Yaskawa INFORM job: test1_robodk.jbi

/JOB
//NAME Hexagon
//POS
///NPOS 620,0,0,0,0,0
///TOOL 9
///POSTYPE PULSE
///PULSE
C00000=-4,42,-30,0,-18,-176
C00001=-4,48,-28,0,-14,-176
C00002=-1,49,-25,0,-16,-179
C00003=-1,52,-18,0,-19,-179
C00004=-4,54,-14,0,-22,-176
C00005=-7,53,-17,0,-20,-173
C00006=-7,50,-24,0,-16,-173
C00007=-4,48,-28,0,-14,-176
C00008=-4,48,-28,0,-14,-176
C00009=-4,48,-28,0,-14,-176
C00010=-4,48,-28,0,-14,-176
C00011=-1,49,-25,0,-16,-179
C00012=-1,52,-18,0,-19,-179
C00013=-4,54,-15,0,-21,-176
C00014=-7,53,-18,0,-20,-173
C00015=-7,50,-24,0,-16,-173
C00016=-4,48,-28,0,-14,-176
C00017=-4,48,-28,0,-14,-176
C00018=-1,49,-25,0,-16,-179
C00019=-1,49,-25,0,-16,-179
C00020=-1,49,-25,0,-15,-179
C00021=-1,49,-25,0,-16,-179
C00022=-2,49,-26,0,-15,-178
C00023=-2,49,-26,0,-15,-178
C00024=-2,49,-26,0,-15,-178
C00025=-1,50,-25,0,-16,-179
C00026=-1,50,-24,0,-16,-179
C00027=-2,49,-26,0,-15,-178
C00028=-2,49,-26,0,-15,-178
C00029=-2,49,-26,0,-15,-178
C00030=-1,50,-24,0,-16,-179
C00031=-1,50,-24,0,-16,-179
C00032=-3,49,-27,0,-15,-177
C00033=-3,49,-27,0,-15,-177
C00034=-3,49,-27,0,-15,-177
C00035=-1,50,-24,0,-16,-179
C00036=-1,50,-24,0,-16,-179
C00037=-3,48,-27,0,-14,-177
C00038=-3,48,-27,0,-14,-177
C00039=-4,48,-27,0,-14,-176
C00040=-1,50,-23,0,-17,-179
C00041=-1,50,-23,0,-17,-179
C00042=-4,48,-28,0,-14,-176
C00043=-4,48,-28,0,-14,-176
C00044=-4,48,-28,0,-14,-176
C00045=-1,50,-23,0,-17,-179
C00046=-1,50,-23,0,-17,-179
C00047=-4,48,-28,0,-14,-176
C00048=-4,48,-28,0,-14,-176
C00049=-1,50,-22,0,-17,-179
C00050=-1,51,-22,0,-17,-179
C00051=-5,48,-28,0,-14,-175
C00052=-5,48,-28,0,-14,-175
C00053=-1,51,-22,0,-17,-179
C00054=-1,51,-22,0,-17,-179
C00055=-5,48,-28,0,-14,-175
C00056=-5,48,-28,0,-14,-175
C00057=-1,51,-22,0,-18,-179
C00058=-1,51,-21,0,-18,-179
C00059=-5,48,-28,0,-14,-175
C00060=-5,48,-27,0,-14,-175
C00061=-1,51,-21,0,-18,-179
C00062=-1,51,-21,0,-18,-179
C00063=-5,48,-27,0,-14,-175
C00064=-5,48,-27,0,-14,-175
C00065=-1,51,-21,0,-18,-179
C00066=-1,51,-21,0,-18,-179
C00067=-5,48,-27,0,-14,-175
C00068=-5,48,-27,0,-14,-175
C00069=-1,51,-20,0,-18,-179
C00070=-1,51,-20,0,-18,-179
C00071=-5,49,-27,0,-14,-175
C00072=-5,49,-27,0,-15,-175
C00073=-1,52,-20,0,-19,-179
C00074=-1,52,-20,0,-19,-179
C00075=-5,49,-27,0,-15,-175
C00076=-5,49,-27,0,-15,-175
C00077=-1,52,-19,0,-19,-179
C00078=-1,52,-19,0,-19,-179
C00079=-5,49,-27,0,-15,-175
C00080=-6,49,-27,0,-15,-174
C00081=-1,52,-19,0,-19,-179
C00082=-1,52,-19,0,-19,-179
C00083=-6,49,-26,0,-15,-174
C00084=-6,49,-26,0,-15,-174
C00085=-1,52,-19,0,-19,-179
C00086=-1,52,-18,0,-19,-179
C00087=-6,49,-26,0,-15,-174
C00088=-6,49,-26,0,-15,-174
C00089=-1,52,-18,0,-19,-179
C00090=-1,52,-18,0,-19,-179
C00091=-6,49,-26,0,-15,-174
C00092=-6,49,-26,0,-15,-174
C00093=-1,52,-18,0,-20,-179
C00094=-1,52,-18,0,-20,-179
C00095=-6,49,-26,0,-15,-174
C00096=-6,49,-26,0,-15,-174
C00097=-2,52,-18,0,-20,-178
C00098=-2,52,-18,0,-20,-178
C00099=-6,49,-26,0,-15,-174
C00100=-6,49,-26,0,-15,-174
C00101=-2,52,-18,0,-20,-178
C00102=-2,52,-18,0,-20,-178
C00103=-6,49,-26,0,-15,-174
C00104=-6,49,-26,0,-15,-174
C00105=-2,53,-18,0,-20,-178
C00106=-2,53,-18,0,-20,-178
C00107=-6,49,-25,0,-15,-174
C00108=-6,49,-25,0,-15,-174
C00109=-2,53,-18,0,-20,-178
C00110=-2,53,-17,0,-20,-178
C00111=-7,49,-25,0,-16,-173
C00112=-7,49,-25,0,-16,-173
C00113=-2,53,-17,0,-20,-178
C00114=-2,53,-17,0,-20,-178
C00115=-7,49,-25,0,-16,-173
C00116=-7,49,-25,0,-16,-173
C00117=-2,53,-17,0,-20,-178
C00118=-2,53,-17,0,-20,-178
C00119=-7,49,-25,0,-16,-173
C00120=-7,49,-25,0,-16,-173
C00121=-2,53,-17,0,-20,-178
C00122=-2,53,-17,0,-20,-178
C00123=-7,49,-25,0,-16,-173
C00124=-7,50,-25,0,-16,-173
C00125=-2,53,-17,0,-20,-178
C00126=-3,53,-17,0,-20,-177
C00127=-7,50,-24,0,-16,-173
C00128=-7,50,-24,0,-16,-173
C00129=-3,53,-17,0,-20,-177
C00130=-3,53,-17,0,-20,-177
C00131=-7,50,-24,0,-16,-173
C00132=-7,50,-24,0,-16,-173
C00133=-3,53,-16,0,-20,-177
C00134=-3,53,-16,0,-21,-177
C00135=-7,50,-24,0,-16,-173
C00136=-7,50,-24,0,-16,-173
C00137=-3,53,-16,0,-21,-177
C00138=-3,53,-16,0,-21,-177
C00139=-7,50,-24,0,-16,-173
C00140=-7,50,-23,0,-17,-173
C00141=-3,53,-16,0,-21,-177
C00142=-3,53,-16,0,-21,-177
C00143=-7,50,-23,0,-17,-173
C00144=-7,50,-23,0,-17,-173
C00145=-3,53,-16,0,-21,-177
C00146=-3,53,-16,0,-21,-177
C00147=-7,50,-23,0,-17,-173
C00148=-7,50,-22,0,-17,-173
C00149=-3,53,-16,0,-21,-177
C00150=-3,53,-16,0,-21,-177
C00151=-7,51,-22,0,-17,-173
C00152=-7,51,-22,0,-17,-173
C00153=-3,53,-16,0,-21,-177
C00154=-3,53,-15,0,-21,-177
C00155=-7,51,-22,0,-17,-173
C00156=-7,51,-22,0,-18,-173
C00157=-3,54,-15,0,-21,-177
C00158=-4,54,-15,0,-21,-176
C00159=-7,51,-21,0,-18,-173
C00160=-7,51,-21,0,-18,-173
C00161=-4,54,-15,0,-21,-176
C00162=-4,54,-15,0,-21,-176
C00163=-7,51,-21,0,-18,-173
C00164=-7,51,-21,0,-18,-173
C00165=-4,54,-15,0,-21,-176
C00166=-4,54,-15,0,-21,-176
C00167=-7,51,-21,0,-18,-173
C00168=-7,51,-20,0,-18,-173
C00169=-4,54,-15,0,-21,-176
C00170=-4,54,-15,0,-21,-176
C00171=-7,51,-20,0,-18,-173
C00172=-7,52,-20,0,-19,-173
C00173=-4,54,-15,0,-21,-176
C00174=-4,54,-15,0,-21,-176
C00175=-4,54,-15,0,-21,-176
C00176=-7,52,-20,0,-19,-173
C00177=-7,52,-19,0,-19,-173
C00178=-5,53,-16,0,-21,-175
C00179=-5,53,-15,0,-21,-175
C00180=-5,53,-16,0,-21,-175
C00181=-7,52,-19,0,-19,-173
C00182=-7,52,-19,0,-19,-173
C00183=-5,53,-16,0,-21,-175
C00184=-5,53,-16,0,-21,-175
C00185=-5,53,-16,0,-21,-175
C00186=-7,52,-19,0,-19,-173
C00187=-7,52,-19,0,-19,-173
C00188=-6,53,-17,0,-20,-174
C00189=-6,53,-17,0,-20,-174
C00190=-6,53,-17,0,-20,-174
C00191=-7,52,-18,0,-19,-173
C00192=-7,52,-18,0,-20,-173
C00193=-6,53,-17,0,-20,-174
C00194=-6,53,-17,0,-20,-174
C00195=-6,53,-17,0,-20,-174
C00196=-7,52,-18,0,-20,-173
C00197=-7,52,-18,0,-20,-173
C00198=-7,53,-18,0,-20,-173
C00199=-7,53,-18,0,-20,-173
C00200=-7,53,-18,0,-20,-173
C00201=-7,52,-18,0,-20,-173
C00202=-4,48,-27,0,-14,-176
C00203=-3,49,-26,0,-15,-177
C00204=-2,49,-25,0,-16,-178
C00205=-1,52,-19,0,-19,-179
C00206=-4,53,-15,0,-21,-176
C00207=-7,52,-18,0,-20,-173
C00208=-7,50,-24,0,-16,-173
C00209=-4,48,-27,0,-14,-176
C00210=-4,48,-28,0,-14,-176
C00211=-3,49,-26,0,-15,-177
C00212=-1,49,-25,0,-16,-179
C00213=-1,52,-19,0,-19,-179
C00214=-4,54,-15,0,-21,-176
C00215=-7,52,-18,0,-20,-173
C00216=-7,50,-24,0,-16,-173
C00217=-4,48,-28,0,-14,-176
C00218=-4,48,-28,0,-14,-176
C00219=-3,49,-26,0,-15,-177
C00220=-1,49,-25,0,-16,-179
C00221=-1,52,-19,0,-19,-179
C00222=-4,54,-15,0,-21,-176
C00223=-7,52,-18,0,-20,-173
C00224=-7,50,-24,0,-16,-173
C00225=-4,48,-28,0,-14,-176
C00226=-4,48,-28,0,-14,-176
C00227=-3,49,-27,0,-15,-177
C00228=-1,49,-25,0,-16,-179
C00229=-1,52,-19,0,-19,-179
C00230=-4,54,-15,0,-21,-176
C00231=-7,52,-18,0,-20,-173
C00232=-7,50,-24,0,-16,-173
C00233=-4,48,-28,0,-14,-176
C00234=-4,48,-28,0,-14,-176
C00235=-4,48,-28,0,-14,-176
C00236=-3,49,-27,0,-15,-177
C00237=-1,49,-25,0,-16,-179
C00238=-1,52,-18,0,-19,-179
C00239=-4,54,-15,0,-22,-176
C00240=-7,52,-18,0,-20,-173
C00241=-7,50,-24,0,-16,-173
C00242=-4,48,-28,0,-14,-176
C00243=-4,48,-28,0,-14,-176
C00244=-4,48,-28,0,-14,-176
C00245=-3,49,-27,0,-15,-177
C00246=-1,49,-25,0,-16,-179
C00247=-1,52,-18,0,-19,-179
C00248=-4,54,-14,0,-22,-176
C00249=-7,53,-18,0,-20,-173
C00250=-7,50,-24,0,-16,-173
C00251=-4,48,-28,0,-14,-176
C00252=-4,48,-28,0,-14,-176
C00253=-4,48,-28,0,-14,-176
C00254=-4,48,-27,0,-14,-176
C00255=-2,49,-25,0,-16,-178
C00256=-2,52,-19,0,-19,-178
C00257=-4,53,-16,0,-21,-176
C00258=-7,52,-18,0,-20,-173
C00259=-7,50,-24,0,-16,-173
C00260=-4,48,-27,0,-14,-176
C00261=-7,50,-24,0,-16,-173
C00262=-7,50,-24,0,-16,-173
C00263=-7,50,-24,0,-16,-173
C00264=-6,50,-24,0,-16,-174
C00265=-6,50,-24,0,-16,-174
C00266=-6,49,-25,0,-16,-174
C00267=-7,50,-23,0,-17,-173
C00268=-7,50,-23,0,-17,-173
C00269=-6,49,-25,0,-16,-174
C00270=-6,49,-25,0,-16,-174
C00271=-6,49,-25,0,-15,-174
C00272=-7,50,-23,0,-17,-173
C00273=-7,50,-23,0,-17,-173
C00274=-6,49,-26,0,-15,-174
C00275=-5,49,-26,0,-15,-175
C00276=-5,49,-26,0,-15,-175
C00277=-7,50,-23,0,-17,-173
C00278=-7,50,-22,0,-17,-173
C00279=-5,49,-26,0,-15,-175
C00280=-5,49,-26,0,-15,-175
C00281=-5,49,-27,0,-15,-175
C00282=-7,50,-22,0,-17,-173
C00283=-7,51,-22,0,-17,-173
C00284=-5,48,-27,0,-15,-175
C00285=-4,48,-27,0,-14,-176
C00286=-4,48,-27,0,-14,-176
C00287=-7,51,-22,0,-18,-173
C00288=-7,51,-22,0,-18,-173
C00289=-4,48,-27,0,-14,-176
C00290=-4,48,-27,0,-14,-176
C00291=-7,51,-21,0,-18,-173
C00292=-7,51,-21,0,-18,-173
C00293=-4,48,-27,0,-15,-176
C00294=-4,48,-27,0,-15,-176
C00295=-7,51,-21,0,-18,-173
C00296=-7,51,-21,0,-18,-173
C00297=-4,49,-27,0,-15,-176
C00298=-4,49,-27,0,-15,-176
C00299=-7,51,-21,0,-18,-173
C00300=-7,51,-20,0,-18,-173
C00301=-4,49,-27,0,-15,-176
C00302=-4,49,-27,0,-15,-176
C00303=-7,51,-20,0,-19,-173
C00304=-7,51,-20,0,-19,-173
C00305=-4,49,-27,0,-15,-176
C00306=-4,49,-27,0,-15,-176
C00307=-7,52,-20,0,-19,-173
C00308=-7,52,-19,0,-19,-173
C00309=-4,49,-26,0,-15,-176
C00310=-3,49,-26,0,-15,-177
C00311=-7,52,-19,0,-19,-173
C00312=-7,52,-19,0,-19,-173
C00313=-3,49,-26,0,-15,-177
C00314=-3,49,-26,0,-15,-177
C00315=-7,52,-19,0,-19,-173
C00316=-6,52,-19,0,-19,-174
C00317=-3,49,-26,0,-15,-177
C00318=-3,49,-26,0,-15,-177
C00319=-6,52,-18,0,-19,-174
C00320=-6,52,-18,0,-20,-174
C00321=-3,49,-26,0,-15,-177
C00322=-3,49,-26,0,-15,-177
C00323=-6,52,-18,0,-20,-174
C00324=-6,52,-18,0,-20,-174
C00325=-3,49,-26,0,-15,-177
C00326=-3,49,-26,0,-15,-177
C00327=-6,52,-18,0,-20,-174
C00328=-6,52,-18,0,-20,-174
C00329=-3,49,-26,0,-15,-177
C00330=-3,49,-26,0,-15,-177
C00331=-6,52,-18,0,-20,-174
C00332=-6,52,-18,0,-20,-174
C00333=-3,49,-26,0,-15,-177
C00334=-3,49,-26,0,-15,-177
C00335=-6,52,-18,0,-20,-174
C00336=-6,52,-18,0,-20,-174
C00337=-2,49,-26,0,-15,-178
C00338=-2,49,-25,0,-15,-178
C00339=-6,52,-18,0,-20,-174
C00340=-6,53,-18,0,-20,-174
C00341=-2,49,-25,0,-15,-178
C00342=-2,49,-25,0,-16,-178
C00343=-6,53,-17,0,-20,-174
C00344=-6,53,-17,0,-20,-174
C00345=-2,49,-25,0,-16,-178
C00346=-2,49,-25,0,-16,-178
C00347=-6,53,-17,0,-20,-174
C00348=-5,53,-17,0,-20,-175
C00349=-2,49,-25,0,-16,-178
C00350=-2,49,-25,0,-16,-178
C00351=-5,53,-17,0,-20,-175
C00352=-5,53,-17,0,-20,-175
C00353=-2,49,-25,0,-16,-178
C00354=-2,49,-25,0,-16,-178
C00355=-5,53,-17,0,-20,-175
C00356=-5,53,-17,0,-20,-175
C00357=-2,49,-25,0,-16,-178
C00358=-2,49,-25,0,-16,-178
C00359=-5,53,-17,0,-20,-175
C00360=-5,53,-17,0,-20,-175
C00361=-2,49,-25,0,-16,-178
C00362=-2,50,-24,0,-16,-178
C00363=-5,53,-17,0,-20,-175
C00364=-5,53,-17,0,-20,-175
C00365=-2,50,-24,0,-16,-178
C00366=-2,50,-24,0,-16,-178
C00367=-5,53,-17,0,-20,-175
C00368=-5,53,-17,0,-20,-175
C00369=-2,50,-24,0,-16,-178
C00370=-2,50,-24,0,-17,-178
C00371=-5,53,-17,0,-21,-175
C00372=-5,53,-16,0,-21,-175
C00373=-2,50,-23,0,-17,-178
C00374=-2,50,-23,0,-17,-178
C00375=-5,53,-16,0,-21,-175
C00376=-5,53,-16,0,-21,-175
C00377=-2,50,-23,0,-17,-178
C00378=-2,50,-23,0,-17,-178
C00379=-4,53,-16,0,-21,-176
C00380=-4,53,-16,0,-21,-176
C00381=-2,50,-22,0,-17,-178
C00382=-2,50,-22,0,-17,-178
C00383=-4,53,-16,0,-21,-176
C00384=-4,53,-16,0,-21,-176
C00385=-2,51,-22,0,-17,-178
C00386=-2,51,-22,0,-18,-178
C00387=-4,53,-16,0,-21,-176
C00388=-4,53,-16,0,-21,-176
C00389=-2,51,-22,0,-18,-178
C00390=-2,51,-21,0,-18,-178
C00391=-4,53,-16,0,-21,-176
C00392=-4,53,-16,0,-21,-176
C00393=-2,51,-21,0,-18,-178
C00394=-2,51,-21,0,-18,-178
C00395=-4,53,-16,0,-21,-176
C00396=-4,53,-16,0,-21,-176
C00397=-4,53,-16,0,-21,-176
C00398=-2,51,-21,0,-18,-178
C00399=-2,51,-21,0,-18,-178
C00400=-3,53,-17,0,-21,-177
C00401=-3,53,-16,0,-21,-177
C00402=-3,53,-17,0,-20,-177
C00403=-2,51,-20,0,-18,-178
C00404=-2,51,-20,0,-18,-178
C00405=-3,53,-17,0,-20,-177
C00406=-3,53,-17,0,-20,-177
C00407=-3,53,-18,0,-20,-177
C00408=-2,51,-20,0,-19,-178
C00409=-2,52,-20,0,-19,-178
C00410=-2,52,-18,0,-20,-178
C00411=-2,52,-18,0,-20,-178
C00412=-2,52,-18,0,-20,-178
C00413=-2,52,-19,0,-19,-178
C00414=-2,52,-19,0,-19,-178
C00415=-2,52,-18,0,-19,-178
C00416=-2,52,-18,0,-19,-178
C00417=-2,52,-19,0,-19,-178
C00418=-2,52,-19,0,-19,-178
C00419=-2,52,-19,0,-19,-178
C00420=-4,48,-28,0,-14,-176
C00421=-4,48,-28,0,-14,-176
C00422=-7,49,-24,0,-16,-173
C00423=-7,52,-18,0,-20,-173
C00424=-4,54,-15,0,-22,-176
C00425=-1,52,-18,0,-20,-179
C00426=-1,49,-25,0,-16,-179
C00427=-4,48,-28,0,-14,-176
C00428=-7,49,-24,0,-16,-173
C00429=-7,52,-18,0,-20,-173
C00430=-4,54,-15,0,-22,-176
C00431=-1,52,-18,0,-20,-179
C00432=-1,49,-25,0,-16,-179
C00433=-4,48,-28,0,-14,-176
C00434=-7,49,-24,0,-16,-173
C00435=-7,52,-18,0,-20,-173
C00436=-4,54,-15,0,-22,-176
C00437=-1,52,-18,0,-20,-179
C00438=-1,49,-25,0,-16,-179
C00439=-4,48,-28,0,-14,-176
C00440=-7,49,-24,0,-16,-173
C00441=-7,52,-18,0,-20,-173
C00442=-4,54,-15,0,-22,-176
C00443=-1,52,-18,0,-20,-179
C00444=-1,49,-25,0,-16,-179
C00445=-4,48,-28,0,-14,-176
C00446=-7,49,-25,0,-16,-173
C00447=-7,52,-18,0,-20,-173
C00448=-4,54,-15,0,-22,-176
C00449=-1,52,-19,0,-20,-179
C00450=-1,49,-25,0,-16,-179
C00451=-4,48,-28,0,-14,-176
C00452=-7,49,-25,0,-16,-173
C00453=-7,52,-18,0,-20,-173
C00454=-4,54,-15,0,-22,-176
C00455=-1,52,-19,0,-20,-179
C00456=-1,49,-25,0,-16,-179
C00457=-4,47,-28,0,-14,-176
C00458=-7,49,-25,0,-16,-173
C00459=-7,52,-18,0,-20,-173
C00460=-4,53,-15,0,-22,-176
C00461=-1,52,-19,0,-20,-179
C00462=-1,49,-25,0,-16,-179
C00463=-4,47,-28,0,-14,-176
C00464=-7,49,-25,0,-16,-173
C00465=-7,52,-18,0,-20,-173
C00466=-4,53,-15,0,-22,-176
C00467=-1,52,-19,0,-20,-179
C00468=-1,49,-25,0,-16,-179
C00469=-4,47,-29,0,-14,-176
C00470=-7,49,-25,0,-16,-173
C00471=-7,52,-18,0,-20,-173
C00472=-4,53,-15,0,-22,-176
C00473=-1,52,-19,0,-20,-179
C00474=-1,49,-26,0,-16,-179
C00475=-4,47,-29,0,-14,-176
C00476=-7,49,-25,0,-16,-173
C00477=-7,52,-18,0,-20,-173
C00478=-4,53,-15,0,-22,-176
C00479=-1,51,-19,0,-20,-179
C00480=-1,48,-26,0,-16,-179
C00481=-4,47,-29,0,-14,-176
C00482=-7,49,-25,0,-16,-173
C00483=-7,52,-18,0,-20,-173
C00484=-4,53,-15,0,-22,-176
C00485=-1,51,-19,0,-20,-179
C00486=-1,48,-26,0,-16,-179
C00487=-4,47,-29,0,-14,-176
C00488=-7,49,-25,0,-17,-173
C00489=-7,52,-18,0,-20,-173
C00490=-4,53,-15,0,-22,-176
C00491=-1,51,-19,0,-20,-179
C00492=-1,48,-26,0,-16,-179
C00493=-4,47,-29,0,-14,-176
C00494=-7,49,-25,0,-17,-173
C00495=-7,52,-18,0,-20,-173
C00496=-4,53,-15,0,-22,-176
C00497=-1,51,-19,0,-20,-179
C00498=-1,48,-26,0,-16,-179
C00499=-4,47,-29,0,-14,-176
C00500=-7,49,-25,0,-17,-173
C00501=-7,52,-18,0,-20,-173
C00502=-4,53,-15,0,-22,-176
C00503=-1,51,-19,0,-20,-179
C00504=-1,48,-26,0,-16,-179
C00505=-4,47,-29,0,-14,-176
C00506=-7,49,-25,0,-17,-173
C00507=-7,52,-18,0,-21,-173
C00508=-4,53,-15,0,-22,-176
C00509=-1,51,-19,0,-20,-179
C00510=-1,48,-26,0,-16,-179
C00511=-4,47,-29,0,-14,-176
C00512=-7,48,-25,0,-17,-173
C00513=-7,51,-18,0,-21,-173
C00514=-4,53,-15,0,-22,-176
C00515=-1,51,-19,0,-20,-179
C00516=-1,48,-26,0,-16,-179
C00517=-4,47,-29,0,-15,-176
C00518=-7,48,-25,0,-17,-173
C00519=-7,51,-18,0,-21,-173
C00520=-4,53,-15,0,-22,-176
C00521=-1,51,-19,0,-20,-179
C00522=-1,48,-26,0,-16,-179
C00523=-4,47,-29,0,-15,-176
C00524=-7,48,-25,0,-17,-173
C00525=-7,51,-18,0,-21,-173
C00526=-4,53,-15,0,-22,-176
C00527=-1,51,-19,0,-20,-179
C00528=-1,48,-26,0,-16,-179
C00529=-4,47,-29,0,-15,-176
C00530=-7,48,-25,0,-17,-173
C00531=-7,51,-18,0,-21,-173
C00532=-4,53,-15,0,-22,-176
C00533=-1,51,-19,0,-20,-179
C00534=-1,48,-26,0,-16,-179
C00535=-4,47,-29,0,-15,-176
C00536=-7,48,-25,0,-17,-173
C00537=-7,51,-18,0,-21,-173
C00538=-4,53,-15,0,-22,-176
C00539=-1,51,-19,0,-20,-179
C00540=-1,48,-26,0,-16,-179
C00541=-4,46,-29,0,-15,-176
C00542=-7,48,-25,0,-17,-173
C00543=-7,51,-18,0,-21,-173
C00544=-4,53,-15,0,-22,-176
C00545=-1,51,-19,0,-20,-179
C00546=-1,48,-26,0,-16,-179
C00547=-4,46,-29,0,-15,-176
C00548=-7,48,-25,0,-17,-173
C00549=-7,51,-18,0,-21,-173
C00550=-4,52,-15,0,-22,-176
C00551=-1,51,-19,0,-20,-179
C00552=-1,48,-26,0,-17,-179
C00553=-4,46,-29,0,-15,-176
C00554=-7,48,-25,0,-17,-173
C00555=-7,51,-18,0,-21,-173
C00556=-4,52,-15,0,-23,-176
C00557=-1,51,-19,0,-20,-179
C00558=-1,48,-26,0,-17,-179
C00559=-4,46,-29,0,-15,-176
C00560=-7,48,-25,0,-17,-173
C00561=-7,51,-18,0,-21,-173
C00562=-4,52,-15,0,-23,-176
C00563=-1,51,-19,0,-20,-179
C00564=-1,47,-26,0,-17,-179
C00565=-4,46,-29,0,-15,-176
C00566=-7,48,-25,0,-17,-173
C00567=-7,51,-18,0,-21,-173
C00568=-4,52,-15,0,-23,-176
C00569=-1,50,-19,0,-20,-179
C00570=-1,47,-26,0,-17,-179
C00571=-4,46,-29,0,-15,-176
C00572=-7,48,-25,0,-17,-173
C00573=-7,51,-18,0,-21,-173
C00574=-4,52,-15,0,-23,-176
C00575=-1,50,-19,0,-21,-179
C00576=-1,47,-26,0,-17,-179
C00577=-4,46,-29,0,-15,-176
C00578=-7,48,-25,0,-17,-173
C00579=-7,51,-18,0,-21,-173
C00580=-4,52,-15,0,-23,-176
C00581=-1,50,-19,0,-21,-179
C00582=-1,47,-26,0,-17,-179
C00583=-4,46,-29,0,-15,-176
C00584=-7,48,-25,0,-17,-173
C00585=-7,51,-18,0,-21,-173
C00586=-4,52,-15,0,-23,-176
C00587=-1,50,-19,0,-21,-179
C00588=-1,47,-26,0,-17,-179
C00589=-4,46,-29,0,-15,-176
C00590=-7,48,-25,0,-17,-173
C00591=-7,51,-18,0,-21,-173
C00592=-4,52,-15,0,-23,-176
C00593=-1,50,-19,0,-21,-179
C00594=-1,47,-26,0,-17,-179
C00595=-4,46,-29,0,-15,-176
C00596=-7,47,-25,0,-17,-173
C00597=-7,51,-18,0,-21,-173
C00598=-4,52,-15,0,-23,-176
C00599=-1,50,-19,0,-21,-179
C00600=-1,47,-26,0,-17,-179
C00601=-4,46,-29,0,-15,-176
C00602=-7,47,-25,0,-17,-173
C00603=-7,50,-18,0,-21,-173
C00604=-4,52,-15,0,-23,-176
C00605=-1,50,-19,0,-21,-179
C00606=-1,47,-26,0,-17,-179
C00607=-4,46,-29,0,-15,-176
C00608=-7,47,-25,0,-17,-173
C00609=-7,50,-18,0,-21,-173
C00610=-4,52,-15,0,-23,-176
C00611=-1,50,-19,0,-21,-179
C00612=-1,47,-26,0,-17,-179
C00613=-4,46,-29,0,-15,-176
C00614=-7,47,-25,0,-17,-173
C00615=-7,50,-18,0,-21,-173
C00616=-4,52,-15,0,-23,-176
C00617=-1,50,-19,0,-21,-179
C00618=-1,47,-26,0,-17,-179
C00619=-1,41,-28,0,-21,-179
//INST
///DATE 2024/04/09 21:09
///COMM Generated using RoboDK
///ATTR SC,RW
///GROUP1 RB1
NOP
'Program generated by RoboDK v
'5.6.7 for Yaskawa GP88 on 09/
'04/2024 21:09:49
'Using nominal kinematics.
CALL JOB:M_RunCo
CALL JOB:M_RunCo
CALL JOB:M_RunCo
CALL JOB:M_RunCo
CALL JOB:Extrude
CALL JOB:Extrude
CALL JOB:M_RunCo
'Using Change Frame (targets w
'rt base):
'1000.8,-608.5,-540.0,0.0,0.0,
'0.0
'Tool Set Tool should be close
' to:
'0.0,0.0,0.0,0.0,0.0,0.0
MOVJ C00000 VJ=50.00 PL=1
MOVL C00001 V=1000.0 PL=1
CALL JOB:Extrude
MOVL C00002 V=1000.0 PL=1
CALL JOB:Extrude
MOVL C00003 V=1000.0 PL=1
CALL JOB:Extrude
MOVL C00004 V=1000.0 PL=1
CALL JOB:Extrude
MOVL C00005 V=1000.0 PL=1
CALL JOB:Extrude
MOVL C00006 V=1000.0 PL=1
CALL JOB:Extrude
MOVL C00007 V=1000.0 PL=1
MOVL C00008 V=1000.0 PL=1
MOVL C00009 V=1000.0 PL=1
MOVL C00010 V=1000.0 PL=1
CALL JOB:Extrude
MOVL C00011 V=120.0 PL=1
CALL JOB:Extrude
MOVL C00012 V=120.0 PL=1
CALL JOB:Extrude
MOVL C00013 V=120.0 PL=1
CALL JOB:Extrude
MOVL C00014 V=120.0 PL=1
CALL JOB:Extrude
MOVL C00015 V=120.0 PL=1
CALL JOB:Extrude
MOVL C00016 V=120.0 PL=1
MOVL C00017 V=1000.0 PL=1
MOVL C00018 V=1000.0 PL=1
CALL JOB:Extrude
MOVL C00019 V=120.0 PL=1
MOVL C00020 V=120.0 PL=1
MOVL C00021 V=1000.0 PL=1
CALL JOB:Extrude
MOVL C00022 V=120.0 PL=1
MOVL C00023 V=120.0 PL=1
MOVL C00024 V=1000.0 PL=1
CALL JOB:Extrude
MOVL C00025 V=120.0 PL=1
MOVL C00026 V=1000.0 PL=1
CALL JOB:Extrude
MOVL C00027 V=120.0 PL=1
MOVL C00028 V=120.0 PL=1
MOVL C00029 V=1000.0 PL=1
CALL JOB:Extrude
MOVL C00030 V=120.0 PL=1
MOVL C00031 V=1000.0 PL=1
CALL JOB:Extrude
MOVL C00032 V=120.0 PL=1
MOVL C00033 V=120.0 PL=1
MOVL C00034 V=1000.0 PL=1
CALL JOB:Extrude
MOVL C00035 V=120.0 PL=1
MOVL C00036 V=1000.0 PL=1
CALL JOB:Extrude
MOVL C00037 V=120.0 PL=1
MOVL C00038 V=120.0 PL=1
MOVL C00039 V=1000.0 PL=1
CALL JOB:Extrude
MOVL C00040 V=120.0 PL=1
MOVL C00041 V=1000.0 PL=1
CALL JOB:Extrude
MOVL C00042 V=120.0 PL=1
MOVL C00043 V=120.0 PL=1
MOVL C00044 V=1000.0 PL=1
CALL JOB:Extrude
MOVL C00045 V=120.0 PL=1
MOVL C00046 V=1000.0 PL=1
CALL JOB:Extrude
MOVL C00047 V=120.0 PL=1
MOVL C00048 V=1000.0 PL=1
CALL JOB:Extrude
MOVL C00049 V=120.0 PL=1
MOVL C00050 V=1000.0 PL=1
CALL JOB:Extrude
MOVL C00051 V=120.0 PL=1
MOVL C00052 V=1000.0 PL=1
CALL JOB:Extrude
MOVL C00053 V=120.0 PL=1
MOVL C00054 V=1000.0 PL=1
CALL JOB:Extrude
MOVL C00055 V=120.0 PL=1
MOVL C00056 V=1000.0 PL=1
CALL JOB:Extrude
MOVL C00057 V=120.0 PL=1
MOVL C00058 V=1000.0 PL=1
CALL JOB:Extrude
MOVL C00059 V=120.0 PL=1
MOVL C00060 V=1000.0 PL=1
CALL JOB:Extrude
MOVL C00061 V=120.0 PL=1
MOVL C00062 V=1000.0 PL=1
CALL JOB:Extrude
MOVL C00063 V=120.0 PL=1
MOVL C00064 V=1000.0 PL=1
CALL JOB:Extrude
MOVL C00065 V=120.0 PL=1
MOVL C00066 V=1000.0 PL=1
CALL JOB:Extrude
MOVL C00067 V=120.0 PL=1
MOVL C00068 V=1000.0 PL=1
CALL JOB:Extrude
MOVL C00069 V=120.0 PL=1
MOVL C00070 V=1000.0 PL=1
CALL JOB:Extrude
MOVL C00071 V=120.0 PL=1
MOVL C00072 V=1000.0 PL=1
CALL JOB:Extrude
MOVL C00073 V=120.0 PL=1
MOVL C00074 V=1000.0 PL=1
CALL JOB:Extrude
MOVL C00075 V=120.0 PL=1
MOVL C00076 V=1000.0 PL=1
CALL JOB:Extrude
MOVL C00077 V=120.0 PL=1
MOVL C00078 V=1000.0 PL=1
CALL JOB:Extrude
MOVL C00079 V=120.0 PL=1
MOVL C00080 V=1000.0 PL=1
CALL JOB:Extrude
MOVL C00081 V=120.0 PL=1
MOVL C00082 V=1000.0 PL=1
CALL JOB:Extrude
MOVL C00083 V=120.0 PL=1
MOVL C00084 V=1000.0 PL=1
CALL JOB:Extrude
MOVL C00085 V=120.0 PL=1
MOVL C00086 V=1000.0 PL=1
CALL JOB:Extrude
CALL JOB:Extrude
MOVL C00087 V=120.0 PL=1
MOVL C00088 V=1000.0 PL=1
CALL JOB:Extrude
MOVL C00089 V=120.0 PL=1
MOVL C00090 V=1000.0 PL=1
CALL JOB:Extrude
MOVL C00091 V=120.0 PL=1
MOVL C00092 V=1000.0 PL=1
CALL JOB:Extrude
MOVL C00093 V=120.0 PL=1
MOVL C00094 V=1000.0 PL=1
CALL JOB:Extrude
MOVL C00095 V=120.0 PL=1
MOVL C00096 V=1000.0 PL=1
CALL JOB:Extrude
MOVL C00097 V=120.0 PL=1
MOVL C00098 V=1000.0 PL=1
CALL JOB:Extrude
MOVL C00099 V=120.0 PL=1
MOVL C00100 V=1000.0 PL=1
CALL JOB:Extrude
MOVL C00101 V=120.0 PL=1
MOVL C00102 V=1000.0 PL=1
CALL JOB:Extrude
MOVL C00103 V=120.0 PL=1
MOVL C00104 V=1000.0 PL=1
CALL JOB:Extrude
MOVL C00105 V=120.0 PL=1
MOVL C00106 V=1000.0 PL=1
CALL JOB:Extrude
MOVL C00107 V=120.0 PL=1
MOVL C00108 V=1000.0 PL=1
CALL JOB:Extrude
MOVL C00109 V=120.0 PL=1
MOVL C00110 V=1000.0 PL=1
CALL JOB:Extrude
MOVL C00111 V=120.0 PL=1
MOVL C00112 V=1000.0 PL=1
CALL JOB:Extrude
MOVL C00113 V=120.0 PL=1
MOVL C00114 V=1000.0 PL=1
CALL JOB:Extrude
MOVL C00115 V=120.0 PL=1
MOVL C00116 V=1000.0 PL=1
CALL JOB:Extrude
MOVL C00117 V=120.0 PL=1
MOVL C00118 V=1000.0 PL=1
CALL JOB:Extrude
MOVL C00119 V=120.0 PL=1
MOVL C00120 V=1000.0 PL=1
CALL JOB:Extrude
MOVL C00121 V=120.0 PL=1
MOVL C00122 V=1000.0 PL=1
CALL JOB:Extrude
MOVL C00123 V=120.0 PL=1
MOVL C00124 V=1000.0 PL=1
CALL JOB:Extrude
MOVL C00125 V=120.0 PL=1
MOVL C00126 V=1000.0 PL=1
CALL JOB:Extrude
MOVL C00127 V=120.0 PL=1
MOVL C00128 V=1000.0 PL=1
CALL JOB:Extrude
MOVL C00129 V=120.0 PL=1
MOVL C00130 V=1000.0 PL=1
CALL JOB:Extrude
MOVL C00131 V=120.0 PL=1
MOVL C00132 V=1000.0 PL=1
CALL JOB:Extrude
MOVL C00133 V=120.0 PL=1
MOVL C00134 V=1000.0 PL=1
CALL JOB:Extrude
MOVL C00135 V=120.0 PL=1
MOVL C00136 V=1000.0 PL=1
CALL JOB:Extrude
MOVL C00137 V=120.0 PL=1
MOVL C00138 V=1000.0 PL=1
CALL JOB:Extrude
MOVL C00139 V=120.0 PL=1
MOVL C00140 V=1000.0 PL=1
CALL JOB:Extrude
CALL JOB:Extrude
MOVL C00141 V=120.0 PL=1
MOVL C00142 V=1000.0 PL=1
CALL JOB:Extrude
MOVL C00143 V=120.0 PL=1
MOVL C00144 V=1000.0 PL=1
CALL JOB:Extrude
MOVL C00145 V=120.0 PL=1
MOVL C00146 V=1000.0 PL=1
CALL JOB:Extrude
MOVL C00147 V=120.0 PL=1
MOVL C00148 V=1000.0 PL=1
CALL JOB:Extrude
MOVL C00149 V=120.0 PL=1
MOVL C00150 V=1000.0 PL=1
CALL JOB:Extrude
MOVL C00151 V=120.0 PL=1
MOVL C00152 V=1000.0 PL=1
CALL JOB:Extrude
MOVL C00153 V=120.0 PL=1
MOVL C00154 V=1000.0 PL=1
CALL JOB:Extrude
MOVL C00155 V=120.0 PL=1
MOVL C00156 V=1000.0 PL=1
CALL JOB:Extrude
MOVL C00157 V=120.0 PL=1
MOVL C00158 V=1000.0 PL=1
CALL JOB:Extrude
MOVL C00159 V=120.0 PL=1
MOVL C00160 V=1000.0 PL=1
CALL JOB:Extrude
MOVL C00161 V=120.0 PL=1
MOVL C00162 V=1000.0 PL=1
CALL JOB:Extrude
MOVL C00163 V=120.0 PL=1
MOVL C00164 V=1000.0 PL=1
CALL JOB:Extrude
MOVL C00165 V=120.0 PL=1
MOVL C00166 V=1000.0 PL=1
CALL JOB:Extrude
MOVL C00167 V=120.0 PL=1
MOVL C00168 V=1000.0 PL=1
CALL JOB:Extrude
MOVL C00169 V=120.0 PL=1
MOVL C00170 V=1000.0 PL=1
CALL JOB:Extrude
MOVL C00171 V=120.0 PL=1
MOVL C00172 V=1000.0 PL=1
CALL JOB:Extrude
MOVL C00173 V=120.0 PL=1
MOVL C00174 V=120.0 PL=1
MOVL C00175 V=1000.0 PL=1
CALL JOB:Extrude
MOVL C00176 V=120.0 PL=1
MOVL C00177 V=1000.0 PL=1
CALL JOB:Extrude
MOVL C00178 V=120.0 PL=1
MOVL C00179 V=120.0 PL=1
MOVL C00180 V=1000.0 PL=1
CALL JOB:Extrude
MOVL C00181 V=120.0 PL=1
MOVL C00182 V=1000.0 PL=1
CALL JOB:Extrude
MOVL C00183 V=120.0 PL=1
MOVL C00184 V=120.0 PL=1
MOVL C00185 V=1000.0 PL=1
CALL JOB:Extrude
MOVL C00186 V=120.0 PL=1
MOVL C00187 V=1000.0 PL=1
CALL JOB:Extrude
MOVL C00188 V=120.0 PL=1
MOVL C00189 V=120.0 PL=1
MOVL C00190 V=1000.0 PL=1
CALL JOB:Extrude
MOVL C00191 V=120.0 PL=1
MOVL C00192 V=1000.0 PL=1
CALL JOB:Extrude
MOVL C00193 V=120.0 PL=1
MOVL C00194 V=120.0 PL=1
MOVL C00195 V=1000.0 PL=1
CALL JOB:Extrude
MOVL C00196 V=120.0 PL=1
MOVL C00197 V=1000.0 PL=1
CALL JOB:Extrude
MOVL C00198 V=120.0 PL=1
MOVL C00199 V=120.0 PL=1
MOVL C00200 V=1000.0 PL=1
MOVL C00201 V=10.0 PL=1
MOVL C00202 V=120.0 PL=1
CALL JOB:Extrude
MOVL C00203 V=120.0 PL=1
CALL JOB:Extrude
MOVL C00204 V=120.0 PL=1
CALL JOB:Extrude
MOVL C00205 V=120.0 PL=1
CALL JOB:Extrude
MOVL C00206 V=120.0 PL=1
CALL JOB:Extrude
MOVL C00207 V=120.0 PL=1
CALL JOB:Extrude
MOVL C00208 V=120.0 PL=1
CALL JOB:Extrude
MOVL C00209 V=120.0 PL=1
MOVL C00210 V=1000.0 PL=1
CALL JOB:Extrude
MOVL C00211 V=120.0 PL=1
CALL JOB:Extrude
MOVL C00212 V=120.0 PL=1
CALL JOB:Extrude
MOVL C00213 V=120.0 PL=1
CALL JOB:Extrude
MOVL C00214 V=120.0 PL=1
CALL JOB:Extrude
MOVL C00215 V=120.0 PL=1
CALL JOB:Extrude
MOVL C00216 V=120.0 PL=1
CALL JOB:Extrude
MOVL C00217 V=120.0 PL=1
MOVL C00218 V=1000.0 PL=1
CALL JOB:Extrude
MOVL C00219 V=120.0 PL=1
CALL JOB:Extrude
MOVL C00220 V=120.0 PL=1
CALL JOB:Extrude
MOVL C00221 V=120.0 PL=1
CALL JOB:Extrude
MOVL C00222 V=120.0 PL=1
CALL JOB:Extrude
MOVL C00223 V=120.0 PL=1
CALL JOB:Extrude
MOVL C00224 V=120.0 PL=1
CALL JOB:Extrude
MOVL C00225 V=120.0 PL=1
MOVL C00226 V=1000.0 PL=1
CALL JOB:Extrude
MOVL C00227 V=120.0 PL=1
CALL JOB:Extrude
MOVL C00228 V=120.0 PL=1
CALL JOB:Extrude
MOVL C00229 V=120.0 PL=1
CALL JOB:Extrude
CALL JOB:Extrude
MOVL C00230 V=120.0 PL=1
CALL JOB:Extrude
MOVL C00231 V=120.0 PL=1
CALL JOB:Extrude
MOVL C00232 V=120.0 PL=1
CALL JOB:Extrude
MOVL C00233 V=120.0 PL=1
MOVL C00234 V=1000.0 PL=1
MOVL C00235 V=1000.0 PL=1
CALL JOB:Extrude
MOVL C00236 V=120.0 PL=1
CALL JOB:Extrude
MOVL C00237 V=120.0 PL=1
CALL JOB:Extrude
MOVL C00238 V=120.0 PL=1
CALL JOB:Extrude
MOVL C00239 V=120.0 PL=1
CALL JOB:Extrude
MOVL C00240 V=120.0 PL=1
CALL JOB:Extrude
MOVL C00241 V=120.0 PL=1
CALL JOB:Extrude
MOVL C00242 V=120.0 PL=1
MOVL C00243 V=1000.0 PL=1
MOVL C00244 V=1000.0 PL=1
CALL JOB:Extrude
MOVL C00245 V=120.0 PL=1
CALL JOB:Extrude
MOVL C00246 V=120.0 PL=1
CALL JOB:Extrude
MOVL C00247 V=120.0 PL=1
CALL JOB:Extrude
MOVL C00248 V=120.0 PL=1
CALL JOB:Extrude
MOVL C00249 V=120.0 PL=1
CALL JOB:Extrude
MOVL C00250 V=120.0 PL=1
CALL JOB:Extrude
MOVL C00251 V=120.0 PL=1
MOVL C00252 V=1000.0 PL=1
MOVL C00253 V=1000.0 PL=1
MOVL C00254 V=1000.0 PL=1
CALL JOB:Extrude
MOVL C00255 V=120.0 PL=1
CALL JOB:Extrude
MOVL C00256 V=120.0 PL=1
CALL JOB:Extrude
MOVL C00257 V=120.0 PL=1
CALL JOB:Extrude
MOVL C00258 V=120.0 PL=1
CALL JOB:Extrude
MOVL C00259 V=120.0 PL=1
CALL JOB:Extrude
MOVL C00260 V=120.0 PL=1
MOVL C00261 V=1000.0 PL=1
CALL JOB:Extrude
MOVL C00262 V=120.0 PL=1
MOVL C00263 V=1000.0 PL=1
CALL JOB:Extrude
MOVL C00264 V=120.0 PL=1
MOVL C00265 V=120.0 PL=1
MOVL C00266 V=1000.0 PL=1
CALL JOB:Extrude
MOVL C00267 V=120.0 PL=1
MOVL C00268 V=1000.0 PL=1
CALL JOB:Extrude
MOVL C00269 V=120.0 PL=1
MOVL C00270 V=120.0 PL=1
MOVL C00271 V=1000.0 PL=1
CALL JOB:Extrude
MOVL C00272 V=120.0 PL=1
MOVL C00273 V=1000.0 PL=1
CALL JOB:Extrude
MOVL C00274 V=120.0 PL=1
MOVL C00275 V=120.0 PL=1
MOVL C00276 V=1000.0 PL=1
CALL JOB:Extrude
MOVL C00277 V=120.0 PL=1
MOVL C00278 V=1000.0 PL=1
CALL JOB:Extrude
MOVL C00279 V=120.0 PL=1
MOVL C00280 V=120.0 PL=1
MOVL C00281 V=1000.0 PL=1
CALL JOB:Extrude
MOVL C00282 V=120.0 PL=1
MOVL C00283 V=1000.0 PL=1
CALL JOB:Extrude
MOVL C00284 V=120.0 PL=1
MOVL C00285 V=120.0 PL=1
MOVL C00286 V=1000.0 PL=1
CALL JOB:Extrude
MOVL C00287 V=120.0 PL=1
MOVL C00288 V=1000.0 PL=1
CALL JOB:Extrude
MOVL C00289 V=120.0 PL=1
MOVL C00290 V=1000.0 PL=1
CALL JOB:Extrude
MOVL C00291 V=120.0 PL=1
MOVL C00292 V=1000.0 PL=1
CALL JOB:Extrude
MOVL C00293 V=120.0 PL=1
MOVL C00294 V=1000.0 PL=1
CALL JOB:Extrude
MOVL C00295 V=120.0 PL=1
MOVL C00296 V=1000.0 PL=1
CALL JOB:Extrude
MOVL C00297 V=120.0 PL=1
MOVL C00298 V=1000.0 PL=1
CALL JOB:Extrude
MOVL C00299 V=120.0 PL=1
MOVL C00300 V=1000.0 PL=1
CALL JOB:Extrude
MOVL C00301 V=120.0 PL=1
MOVL C00302 V=1000.0 PL=1
CALL JOB:Extrude
MOVL C00303 V=120.0 PL=1
MOVL C00304 V=1000.0 PL=1
CALL JOB:Extrude
MOVL C00305 V=120.0 PL=1
MOVL C00306 V=1000.0 PL=1
CALL JOB:Extrude
MOVL C00307 V=120.0 PL=1
MOVL C00308 V=1000.0 PL=1
CALL JOB:Extrude
MOVL C00309 V=120.0 PL=1
MOVL C00310 V=1000.0 PL=1
CALL JOB:Extrude
MOVL C00311 V=120.0 PL=1
MOVL C00312 V=1000.0 PL=1
CALL JOB:Extrude
MOVL C00313 V=120.0 PL=1
MOVL C00314 V=1000.0 PL=1
CALL JOB:Extrude
MOVL C00315 V=120.0 PL=1
MOVL C00316 V=1000.0 PL=1
CALL JOB:Extrude
MOVL C00317 V=120.0 PL=1
MOVL C00318 V=1000.0 PL=1
CALL JOB:Extrude
MOVL C00319 V=120.0 PL=1
MOVL C00320 V=1000.0 PL=1
CALL JOB:Extrude
CALL JOB:Extrude
MOVL C00321 V=120.0 PL=1
MOVL C00322 V=1000.0 PL=1
CALL JOB:Extrude
MOVL C00323 V=120.0 PL=1
MOVL C00324 V=1000.0 PL=1
CALL JOB:Extrude
MOVL C00325 V=120.0 PL=1
MOVL C00326 V=1000.0 PL=1
CALL JOB:Extrude
MOVL C00327 V=120.0 PL=1
MOVL C00328 V=1000.0 PL=1
CALL JOB:Extrude
MOVL C00329 V=120.0 PL=1
MOVL C00330 V=1000.0 PL=1
CALL JOB:Extrude
MOVL C00331 V=120.0 PL=1
MOVL C00332 V=1000.0 PL=1
CALL JOB:Extrude
MOVL C00333 V=120.0 PL=1
MOVL C00334 V=1000.0 PL=1
CALL JOB:Extrude
MOVL C00335 V=120.0 PL=1
MOVL C00336 V=1000.0 PL=1
CALL JOB:Extrude
MOVL C00337 V=120.0 PL=1
MOVL C00338 V=1000.0 PL=1
CALL JOB:Extrude
MOVL C00339 V=120.0 PL=1
MOVL C00340 V=1000.0 PL=1
CALL JOB:Extrude
MOVL C00341 V=120.0 PL=1
MOVL C00342 V=1000.0 PL=1
CALL JOB:Extrude
MOVL C00343 V=120.0 PL=1
MOVL C00344 V=1000.0 PL=1
CALL JOB:Extrude
MOVL C00345 V=120.0 PL=1
MOVL C00346 V=1000.0 PL=1
CALL JOB:Extrude
MOVL C00347 V=120.0 PL=1
MOVL C00348 V=1000.0 PL=1
CALL JOB:Extrude
MOVL C00349 V=120.0 PL=1
MOVL C00350 V=1000.0 PL=1
CALL JOB:Extrude
MOVL C00351 V=120.0 PL=1
MOVL C00352 V=1000.0 PL=1
CALL JOB:Extrude
MOVL C00353 V=120.0 PL=1
MOVL C00354 V=1000.0 PL=1
CALL JOB:Extrude
MOVL C00355 V=120.0 PL=1
MOVL C00356 V=1000.0 PL=1
CALL JOB:Extrude
MOVL C00357 V=120.0 PL=1
MOVL C00358 V=1000.0 PL=1
CALL JOB:Extrude
MOVL C00359 V=120.0 PL=1
MOVL C00360 V=1000.0 PL=1
CALL JOB:Extrude
MOVL C00361 V=120.0 PL=1
MOVL C00362 V=1000.0 PL=1
CALL JOB:Extrude
MOVL C00363 V=120.0 PL=1
MOVL C00364 V=1000.0 PL=1
CALL JOB:Extrude
MOVL C00365 V=120.0 PL=1
MOVL C00366 V=1000.0 PL=1
CALL JOB:Extrude
MOVL C00367 V=120.0 PL=1
MOVL C00368 V=1000.0 PL=1
CALL JOB:Extrude
MOVL C00369 V=120.0 PL=1
MOVL C00370 V=1000.0 PL=1
CALL JOB:Extrude
MOVL C00371 V=120.0 PL=1
MOVL C00372 V=1000.0 PL=1
CALL JOB:Extrude
MOVL C00373 V=120.0 PL=1
MOVL C00374 V=1000.0 PL=1
CALL JOB:Extrude
MOVL C00375 V=120.0 PL=1
MOVL C00376 V=1000.0 PL=1
CALL JOB:Extrude
MOVL C00377 V=120.0 PL=1
MOVL C00378 V=1000.0 PL=1
CALL JOB:Extrude
MOVL C00379 V=120.0 PL=1
MOVL C00380 V=1000.0 PL=1
CALL JOB:Extrude
MOVL C00381 V=120.0 PL=1
MOVL C00382 V=1000.0 PL=1
CALL JOB:Extrude
MOVL C00383 V=120.0 PL=1
MOVL C00384 V=1000.0 PL=1
CALL JOB:Extrude
CALL JOB:Extrude
MOVL C00385 V=120.0 PL=1
MOVL C00386 V=1000.0 PL=1
CALL JOB:Extrude
MOVL C00387 V=120.0 PL=1
MOVL C00388 V=1000.0 PL=1
CALL JOB:Extrude
MOVL C00389 V=120.0 PL=1
MOVL C00390 V=1000.0 PL=1
CALL JOB:Extrude
MOVL C00391 V=120.0 PL=1
MOVL C00392 V=1000.0 PL=1
CALL JOB:Extrude
MOVL C00393 V=120.0 PL=1
MOVL C00394 V=1000.0 PL=1
CALL JOB:Extrude
MOVL C00395 V=120.0 PL=1
MOVL C00396 V=120.0 PL=1
MOVL C00397 V=1000.0 PL=1
CALL JOB:Extrude
MOVL C00398 V=120.0 PL=1
MOVL C00399 V=1000.0 PL=1
CALL JOB:Extrude
MOVL C00400 V=120.0 PL=1
MOVL C00401 V=120.0 PL=1
MOVL C00402 V=1000.0 PL=1
CALL JOB:Extrude
MOVL C00403 V=120.0 PL=1
MOVL C00404 V=1000.0 PL=1
CALL JOB:Extrude
MOVL C00405 V=120.0 PL=1
MOVL C00406 V=120.0 PL=1
MOVL C00407 V=1000.0 PL=1
CALL JOB:Extrude
MOVL C00408 V=120.0 PL=1
MOVL C00409 V=1000.0 PL=1
CALL JOB:Extrude
MOVL C00410 V=120.0 PL=1
MOVL C00411 V=120.0 PL=1
MOVL C00412 V=1000.0 PL=1
CALL JOB:Extrude
MOVL C00413 V=120.0 PL=1
MOVL C00414 V=1000.0 PL=1
CALL JOB:Extrude
MOVL C00415 V=120.0 PL=1
MOVL C00416 V=120.0 PL=1
MOVL C00417 V=1000.0 PL=1
CALL JOB:Extrude
MOVL C00418 V=120.0 PL=1
MOVL C00419 V=10.0 PL=1
MOVL C00420 V=120.0 PL=1
MOVL C00421 V=1000.0 PL=1
CALL JOB:Extrude
MOVL C00422 V=120.0 PL=1
CALL JOB:Extrude
MOVL C00423 V=120.0 PL=1
CALL JOB:Extrude
MOVL C00424 V=120.0 PL=1
CALL JOB:Extrude
MOVL C00425 V=120.0 PL=1
CALL JOB:Extrude
MOVL C00426 V=120.0 PL=1
CALL JOB:Extrude
MOVL C00427 V=120.0 PL=1
CALL JOB:Extrude
MOVL C00428 V=120.0 PL=1
CALL JOB:Extrude
MOVL C00429 V=120.0 PL=1
CALL JOB:Extrude
MOVL C00430 V=120.0 PL=1
CALL JOB:Extrude
MOVL C00431 V=120.0 PL=1
CALL JOB:Extrude
MOVL C00432 V=120.0 PL=1
CALL JOB:Extrude
MOVL C00433 V=120.0 PL=1
CALL JOB:Extrude
MOVL C00434 V=109.5 PL=1
CALL JOB:Extrude
MOVL C00435 V=109.5 PL=1
CALL JOB:Extrude
MOVL C00436 V=109.5 PL=1
CALL JOB:Extrude
MOVL C00437 V=109.5 PL=1
CALL JOB:Extrude
MOVL C00438 V=109.5 PL=1
CALL JOB:Extrude
MOVL C00439 V=109.5 PL=1
CALL JOB:Extrude
MOVL C00440 V=109.5 PL=1
CALL JOB:Extrude
MOVL C00441 V=109.5 PL=1
CALL JOB:Extrude
MOVL C00442 V=109.5 PL=1
CALL JOB:Extrude
MOVL C00443 V=109.5 PL=1
CALL JOB:Extrude
MOVL C00444 V=109.5 PL=1
CALL JOB:Extrude
MOVL C00445 V=109.5 PL=1
CALL JOB:Extrude
MOVL C00446 V=109.5 PL=1
CALL JOB:Extrude
MOVL C00447 V=109.5 PL=1
CALL JOB:Extrude
MOVL C00448 V=109.5 PL=1
CALL JOB:Extrude
MOVL C00449 V=109.5 PL=1
CALL JOB:Extrude
MOVL C00450 V=109.5 PL=1
CALL JOB:Extrude
MOVL C00451 V=109.5 PL=1
CALL JOB:Extrude
MOVL C00452 V=109.5 PL=1
CALL JOB:Extrude
MOVL C00453 V=109.5 PL=1
CALL JOB:Extrude
MOVL C00454 V=109.5 PL=1
CALL JOB:Extrude
MOVL C00455 V=109.5 PL=1
CALL JOB:Extrude
MOVL C00456 V=109.5 PL=1
CALL JOB:Extrude
MOVL C00457 V=109.5 PL=1
CALL JOB:Extrude
CALL JOB:Extrude
MOVL C00458 V=109.5 PL=1
CALL JOB:Extrude
MOVL C00459 V=109.5 PL=1
CALL JOB:Extrude
MOVL C00460 V=109.5 PL=1
CALL JOB:Extrude
MOVL C00461 V=109.5 PL=1
CALL JOB:Extrude
MOVL C00462 V=109.5 PL=1
CALL JOB:Extrude
MOVL C00463 V=109.5 PL=1
CALL JOB:Extrude
MOVL C00464 V=109.5 PL=1
CALL JOB:Extrude
MOVL C00465 V=109.5 PL=1
CALL JOB:Extrude
MOVL C00466 V=109.5 PL=1
CALL JOB:Extrude
MOVL C00467 V=109.5 PL=1
CALL JOB:Extrude
MOVL C00468 V=109.5 PL=1
CALL JOB:Extrude
MOVL C00469 V=109.5 PL=1
CALL JOB:Extrude
MOVL C00470 V=109.5 PL=1
CALL JOB:Extrude
MOVL C00471 V=109.5 PL=1
CALL JOB:Extrude
MOVL C00472 V=109.5 PL=1
CALL JOB:Extrude
MOVL C00473 V=109.5 PL=1
CALL JOB:Extrude
MOVL C00474 V=109.5 PL=1
CALL JOB:Extrude
MOVL C00475 V=109.5 PL=1
CALL JOB:Extrude
MOVL C00476 V=109.5 PL=1
CALL JOB:Extrude
MOVL C00477 V=109.5 PL=1
CALL JOB:Extrude
MOVL C00478 V=109.5 PL=1
CALL JOB:Extrude
MOVL C00479 V=109.5 PL=1
CALL JOB:Extrude
MOVL C00480 V=109.5 PL=1
CALL JOB:Extrude
MOVL C00481 V=109.5 PL=1
CALL JOB:Extrude
MOVL C00482 V=109.5 PL=1
CALL JOB:Extrude
MOVL C00483 V=109.5 PL=1
CALL JOB:Extrude
MOVL C00484 V=109.5 PL=1
CALL JOB:Extrude
MOVL C00485 V=109.5 PL=1
CALL JOB:Extrude
MOVL C00486 V=109.5 PL=1
CALL JOB:Extrude
MOVL C00487 V=109.5 PL=1
CALL JOB:Extrude
MOVL C00488 V=109.5 PL=1
CALL JOB:Extrude
MOVL C00489 V=109.5 PL=1
CALL JOB:Extrude
MOVL C00490 V=109.5 PL=1
CALL JOB:Extrude
MOVL C00491 V=109.5 PL=1
CALL JOB:Extrude
MOVL C00492 V=109.5 PL=1
CALL JOB:Extrude
MOVL C00493 V=109.5 PL=1
CALL JOB:Extrude
MOVL C00494 V=109.5 PL=1
CALL JOB:Extrude
MOVL C00495 V=109.5 PL=1
CALL JOB:Extrude
MOVL C00496 V=109.5 PL=1
CALL JOB:Extrude
MOVL C00497 V=109.5 PL=1
CALL JOB:Extrude
MOVL C00498 V=109.5 PL=1
CALL JOB:Extrude
MOVL C00499 V=109.5 PL=1
CALL JOB:Extrude
MOVL C00500 V=109.5 PL=1
CALL JOB:Extrude
MOVL C00501 V=109.5 PL=1
CALL JOB:Extrude
MOVL C00502 V=109.5 PL=1
CALL JOB:Extrude
MOVL C00503 V=109.5 PL=1
CALL JOB:Extrude
CALL JOB:Extrude
MOVL C00504 V=109.5 PL=1
CALL JOB:Extrude
MOVL C00505 V=109.5 PL=1
CALL JOB:Extrude
MOVL C00506 V=109.5 PL=1
CALL JOB:Extrude
MOVL C00507 V=109.5 PL=1
CALL JOB:Extrude
MOVL C00508 V=109.5 PL=1
CALL JOB:Extrude
MOVL C00509 V=109.5 PL=1
CALL JOB:Extrude
MOVL C00510 V=109.5 PL=1
CALL JOB:Extrude
MOVL C00511 V=109.5 PL=1
CALL JOB:Extrude
MOVL C00512 V=109.5 PL=1
CALL JOB:Extrude
MOVL C00513 V=109.5 PL=1
CALL JOB:Extrude
MOVL C00514 V=109.5 PL=1
CALL JOB:Extrude
MOVL C00515 V=109.5 PL=1
CALL JOB:Extrude
MOVL C00516 V=109.5 PL=1
CALL JOB:Extrude
MOVL C00517 V=109.5 PL=1
CALL JOB:Extrude
MOVL C00518 V=109.5 PL=1
CALL JOB:Extrude
MOVL C00519 V=109.5 PL=1
CALL JOB:Extrude
MOVL C00520 V=109.5 PL=1
CALL JOB:Extrude
MOVL C00521 V=109.5 PL=1
CALL JOB:Extrude
MOVL C00522 V=109.5 PL=1
CALL JOB:Extrude
MOVL C00523 V=109.5 PL=1
CALL JOB:Extrude
MOVL C00524 V=109.5 PL=1
CALL JOB:Extrude
MOVL C00525 V=109.5 PL=1
CALL JOB:Extrude
MOVL C00526 V=109.5 PL=1
CALL JOB:Extrude
MOVL C00527 V=109.5 PL=1
CALL JOB:Extrude
MOVL C00528 V=109.5 PL=1
CALL JOB:Extrude
MOVL C00529 V=109.5 PL=1
CALL JOB:Extrude
MOVL C00530 V=109.5 PL=1
CALL JOB:Extrude
MOVL C00531 V=109.5 PL=1
CALL JOB:Extrude
MOVL C00532 V=109.5 PL=1
CALL JOB:Extrude
MOVL C00533 V=109.5 PL=1
CALL JOB:Extrude
MOVL C00534 V=109.5 PL=1
CALL JOB:Extrude
MOVL C00535 V=109.5 PL=1
CALL JOB:Extrude
MOVL C00536 V=109.5 PL=1
CALL JOB:Extrude
MOVL C00537 V=109.5 PL=1
CALL JOB:Extrude
MOVL C00538 V=109.5 PL=1
CALL JOB:Extrude
MOVL C00539 V=109.5 PL=1
CALL JOB:Extrude
MOVL C00540 V=109.5 PL=1
CALL JOB:Extrude
MOVL C00541 V=109.5 PL=1
CALL JOB:Extrude
MOVL C00542 V=109.5 PL=1
CALL JOB:Extrude
MOVL C00543 V=109.5 PL=1
CALL JOB:Extrude
MOVL C00544 V=109.5 PL=1
CALL JOB:Extrude
MOVL C00545 V=109.5 PL=1
CALL JOB:Extrude
MOVL C00546 V=109.5 PL=1
CALL JOB:Extrude
MOVL C00547 V=109.5 PL=1
CALL JOB:Extrude
MOVL C00548 V=109.5 PL=1
CALL JOB:Extrude
MOVL C00549 V=109.5 PL=1
CALL JOB:Extrude
CALL JOB:Extrude
MOVL C00550 V=109.5 PL=1
CALL JOB:Extrude
MOVL C00551 V=109.5 PL=1
CALL JOB:Extrude
MOVL C00552 V=109.5 PL=1
CALL JOB:Extrude
MOVL C00553 V=109.5 PL=1
CALL JOB:Extrude
MOVL C00554 V=109.5 PL=1
CALL JOB:Extrude
MOVL C00555 V=109.5 PL=1
CALL JOB:Extrude
MOVL C00556 V=109.5 PL=1
CALL JOB:Extrude
MOVL C00557 V=109.5 PL=1
CALL JOB:Extrude
MOVL C00558 V=109.5 PL=1
CALL JOB:Extrude
MOVL C00559 V=109.5 PL=1
CALL JOB:Extrude
MOVL C00560 V=109.5 PL=1
CALL JOB:Extrude
MOVL C00561 V=109.5 PL=1
CALL JOB:Extrude
MOVL C00562 V=109.5 PL=1
CALL JOB:Extrude
MOVL C00563 V=109.5 PL=1
CALL JOB:Extrude
MOVL C00564 V=109.5 PL=1
CALL JOB:Extrude
MOVL C00565 V=109.5 PL=1
CALL JOB:Extrude
MOVL C00566 V=109.5 PL=1
CALL JOB:Extrude
MOVL C00567 V=109.5 PL=1
CALL JOB:Extrude
MOVL C00568 V=109.5 PL=1
CALL JOB:Extrude
MOVL C00569 V=109.5 PL=1
CALL JOB:Extrude
MOVL C00570 V=109.5 PL=1
CALL JOB:Extrude
MOVL C00571 V=109.5 PL=1
CALL JOB:Extrude
MOVL C00572 V=109.5 PL=1
CALL JOB:Extrude
MOVL C00573 V=109.5 PL=1
CALL JOB:Extrude
MOVL C00574 V=109.5 PL=1
CALL JOB:Extrude
MOVL C00575 V=109.5 PL=1
CALL JOB:Extrude
MOVL C00576 V=109.5 PL=1
CALL JOB:Extrude
MOVL C00577 V=109.5 PL=1
CALL JOB:Extrude
MOVL C00578 V=109.5 PL=1
CALL JOB:Extrude
MOVL C00579 V=109.5 PL=1
CALL JOB:Extrude
MOVL C00580 V=109.5 PL=1
CALL JOB:Extrude
MOVL C00581 V=109.5 PL=1
CALL JOB:Extrude
MOVL C00582 V=109.5 PL=1
CALL JOB:Extrude
MOVL C00583 V=109.5 PL=1
CALL JOB:Extrude
MOVL C00584 V=109.5 PL=1
CALL JOB:Extrude
MOVL C00585 V=109.5 PL=1
CALL JOB:Extrude
MOVL C00586 V=109.5 PL=1
CALL JOB:Extrude
MOVL C00587 V=109.5 PL=1
CALL JOB:Extrude
MOVL C00588 V=109.5 PL=1
CALL JOB:Extrude
MOVL C00589 V=109.5 PL=1
CALL JOB:Extrude
MOVL C00590 V=109.5 PL=1
CALL JOB:Extrude
MOVL C00591 V=109.5 PL=1
CALL JOB:Extrude
MOVL C00592 V=109.5 PL=1
CALL JOB:Extrude
MOVL C00593 V=109.5 PL=1
CALL JOB:Extrude
MOVL C00594 V=109.5 PL=1
CALL JOB:Extrude
MOVL C00595 V=109.5 PL=1
CALL JOB:Extrude
CALL JOB:Extrude
MOVL C00596 V=109.5 PL=1
CALL JOB:Extrude
MOVL C00597 V=109.5 PL=1
CALL JOB:Extrude
MOVL C00598 V=109.5 PL=1
CALL JOB:Extrude
MOVL C00599 V=109.5 PL=1
CALL JOB:Extrude
MOVL C00600 V=109.5 PL=1
CALL JOB:Extrude
MOVL C00601 V=109.5 PL=1
CALL JOB:Extrude
MOVL C00602 V=109.5 PL=1
CALL JOB:Extrude
MOVL C00603 V=109.5 PL=1
CALL JOB:Extrude
MOVL C00604 V=109.5 PL=1
CALL JOB:Extrude
MOVL C00605 V=109.5 PL=1
CALL JOB:Extrude
MOVL C00606 V=109.5 PL=1
CALL JOB:Extrude
MOVL C00607 V=109.5 PL=1
CALL JOB:Extrude
MOVL C00608 V=109.5 PL=1
CALL JOB:Extrude
MOVL C00609 V=109.5 PL=1
CALL JOB:Extrude
MOVL C00610 V=109.5 PL=1
CALL JOB:Extrude
MOVL C00611 V=109.5 PL=1
CALL JOB:Extrude
MOVL C00612 V=109.5 PL=1
CALL JOB:Extrude
MOVL C00613 V=109.5 PL=1
CALL JOB:Extrude
MOVL C00614 V=109.5 PL=1
CALL JOB:Extrude
MOVL C00615 V=109.5 PL=1
CALL JOB:Extrude
MOVL C00616 V=109.5 PL=1
CALL JOB:Extrude
MOVL C00617 V=109.5 PL=1
MOVL C00618 V=109.5 PL=1
MOVL C00619 V=1000.0 PL=1
CALL JOB:M_RunCo
CALL JOB:M_RunCo
END
